{attribute addProperty BoxType "EL6201-0000-0017"}
{attribute addProperty Id "Slave_28A_DO0BIT10.125217Slave_28A_DO1BIT10.125218Slave_28A_DO2BIT10.125219Slave_28A_DO3BIT10.125220Slave_28B_DO0BIT10.125221Slave_28B_DO1BIT10.125222Slave_28B_DO2BIT10.125223Slave_28B_DO3BIT10.125224"}
{attribute addProperty CRC "3194352330"}
{attribute addProperty SizeInBites "8"}
{attribute addProperty SizeInBytes "1"}
TYPE Slave_28_Outputs_BE65F2CA :
STRUCT
	{attribute addProperty Name "Slave_28A_DO0"}
	Slave_28A_DO0 : BIT;
	{attribute addProperty Name "Slave_28A_DO1"}
	Slave_28A_DO1 : BIT;
	{attribute addProperty Name "Slave_28A_DO2"}
	Slave_28A_DO2 : BIT;
	{attribute addProperty Name "Slave_28A_DO3"}
	Slave_28A_DO3 : BIT;
	{attribute addProperty Name "Slave_28B_DO0"}
	Slave_28B_DO0 : BIT;
	{attribute addProperty Name "Slave_28B_DO1"}
	Slave_28B_DO1 : BIT;
	{attribute addProperty Name "Slave_28B_DO2"}
	Slave_28B_DO2 : BIT;
	{attribute addProperty Name "Slave_28B_DO3"}
	Slave_28B_DO3 : BIT;
END_STRUCT
END_TYPE

(* stored: Version 1.2.0.0, ProductVersion 3.1.4024.9
   DUT Slave_28_Outputs_BE65F2CA: Id {93db19ec-5d63-4692-a5c1-de6002f58c79} *)
